(* PLC project Senza_nome, Sconosciuto Senza_nome 1 *)
(* stored: creationDateTime 2026-06-20T10:48:42, modificationDateTime 2026-06-21T15:30:50 *)

FUNCTION_BLOCK comparison
  VAR_INPUT
    value : INT;
    lowerBound : INT;
    upperBound : INT;
  END_VAR
  VAR_OUTPUT
    output : BOOL;
  END_VAR

            output := (value >= lowerBound) AND (value <= upperBound);
          
END_FUNCTION_BLOCK

PROGRAM program0
  VAR
    boxWeight AT %QW0 : INT;
    boxType AT %QW1 : INT;
    toAddA AT %QW2 : INT;
    toAddB AT %QW3 : INT;
    toAddC AT %QW4 : INT;
    turbineWeight AT %QW5 : INT;
    turbineValidity AT %QX0.0 : BOOL;
  END_VAR
  VAR
    comparison0 : comparison;
    comparison1 : comparison;
  END_VAR

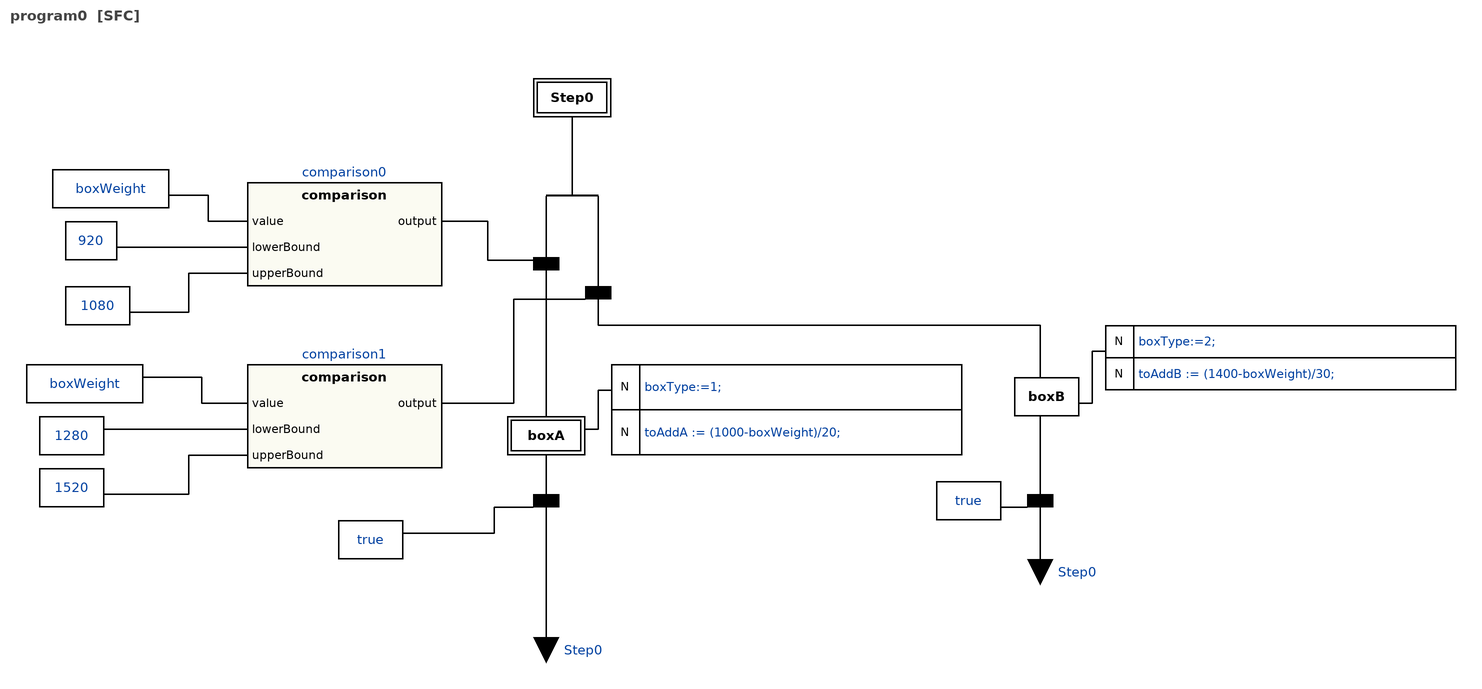
INITIAL_STEP Step0:
  COMPUTE_FUNCTION_BLOCKS(S);
END_STEP
TRANSITION FROM Step0 TO boxA
  := comparison0.output;
END_TRANSITION
TRANSITION FROM Step0 TO boxB
  := comparison1.output;
END_TRANSITION
INITIAL_STEP boxA:
  BOXA_INLINE1(N);
  BOXA_INLINE2(N);
END_STEP
ACTION BOXA_INLINE1:
  boxType:=1;
END_ACTION
ACTION BOXA_INLINE2:
  toAddA := (1000-boxWeight)/20;
END_ACTION
TRANSITION FROM boxA TO Step0
  := true;
END_TRANSITION
STEP boxB:
  BOXB_INLINE3(N);
  BOXB_INLINE4(N);
END_STEP
ACTION BOXB_INLINE3:
  boxType:=2;
END_ACTION
ACTION BOXB_INLINE4:
  toAddB := (1400-boxWeight)/30;
END_ACTION
TRANSITION FROM boxB TO Step0
  := true;
END_TRANSITION
ACTION COMPUTE_FUNCTION_BLOCKS:  (* blocks drawn on the SFC sheet *)
  comparison0(value := boxWeight, lowerBound := 920, upperBound := 1080);
  comparison1(value := boxWeight, lowerBound := 1280, upperBound := 1520);
END_ACTION
END_PROGRAM

CONFIGURATION Config0
  RESOURCE Res0 ON PLC
    TASK task0(INTERVAL := T#20ms, PRIORITY := 0);
    PROGRAM instance0 WITH task0 : program0;
  END_RESOURCE
END_CONFIGURATION
